{attribute 'linkalways'} 
{attribute 'no_explicit_call' := 'This FB is a CLASS and must be accessed using methods or properties'}
{attribute 'enable_dynamic_creation'}
FUNCTION_BLOCK Transition
VAR
	_event : INT;
	_sourceState : I_State;
	_destinationState : I_State;
END_VAR

PROPERTY DestinationState : I_State
GET
DestinationState := _destinationState;
END_GET
END_PROPERTY

PROPERTY Event : INT
GET
Event := _event;
END_GET
END_PROPERTY

METHOD FB_init : BOOL
VAR_INPUT
	bInitRetains : BOOL; // if TRUE, the retain variables are initialized (warm start / cold start)
	bInCopyCode : BOOL;  // if TRUE, the instance afterwards gets moved into the copy code (online change)
	event : INT;
	sourceState : I_State;
	destinationState : I_State;
END_VAR
_event := event;
_sourceState := sourceState;
_destinationState := destinationState;
END_METHOD

PROPERTY SourceState : I_State
GET
SourceState := _sourceState;
END_GET
END_PROPERTY

END_FUNCTION_BLOCK

(* stored: Version 1.1.0.1, ProductVersion 3.1.4024.12
   POU Transition: Id {dc5f1b9e-c438-09f5-22ef-0034eaac9a00}, SpecialFunc None
   Property DestinationState: Id {4993eb70-6edd-053d-1481-92a7d4ccd47a}
   Get Get: Id {011cb777-ebb6-0de5-2327-77b2d0d60d38}
   Property Event: Id {d8bf9cc5-cfbb-0115-09a0-d58ba54880ed}
   Get Get: Id {eae50424-bdd0-0841-3db5-c744f290613e}
   Method FB_init: Id {6efdf76e-b6a7-00cc-3942-2a94fd8de71f}
   Property SourceState: Id {19edc98a-9329-089d-030b-6ae21625bbc5}
   Get Get: Id {e1f63828-71b5-05ab-0468-7fafb6020c6d} *)
